FUNCTION_BLOCK Leg_Model_Mapping_Control
VAR_INPUT
	Model_Leg		: ARRAY [1..18] OF LREAL;			// 模型中的腿编号
END_VAR
VAR_OUTPUT
	Control_Leg		: ARRAY [1..18] OF LREAL;			// 控制程序中的腿编号
END_VAR

Control_Leg[1] 		:= Model_Leg[1];
Control_Leg[2] 		:= Model_Leg[6];
Control_Leg[3] 		:= Model_Leg[5];
Control_Leg[4] 		:= Model_Leg[4];
Control_Leg[5] 		:= Model_Leg[3];
Control_Leg[6] 		:= Model_Leg[2];

END_FUNCTION_BLOCK

(* stored: Version 1.1.0.1, ProductVersion 3.1.4020.12
   POU Leg_Model_Mapping_Control: Id {4d805766-6301-4e45-930b-18b1f845242a}, SpecialFunc None *)
